% RSLogix 500 project traffic_light_rtc.RSS, saved by version 8.30.00.16 %
PROJECT "UNTITLED"    % processor: Bul.1763 MicroLogix 1100 Series A %

PROGRAM FILES
  LAD 2   7 rungs

DATA FILES
  O0 OUTPUT  4 elements
  I1 INPUT  6 elements
  S2 STATUS  66 elements
  B3 BINARY  2 elements
  T4 TIMER  4 elements
  C5 COUNTER  1 elements
  R6 CONTROL  1 elements
  N7 INTEGER  1 elements
  F8 FLOAT  1 elements
  B235   1 elements
  L244   4 elements
  L245   6 elements
  N254   1 elements
  N255   14 elements

LADDER 2
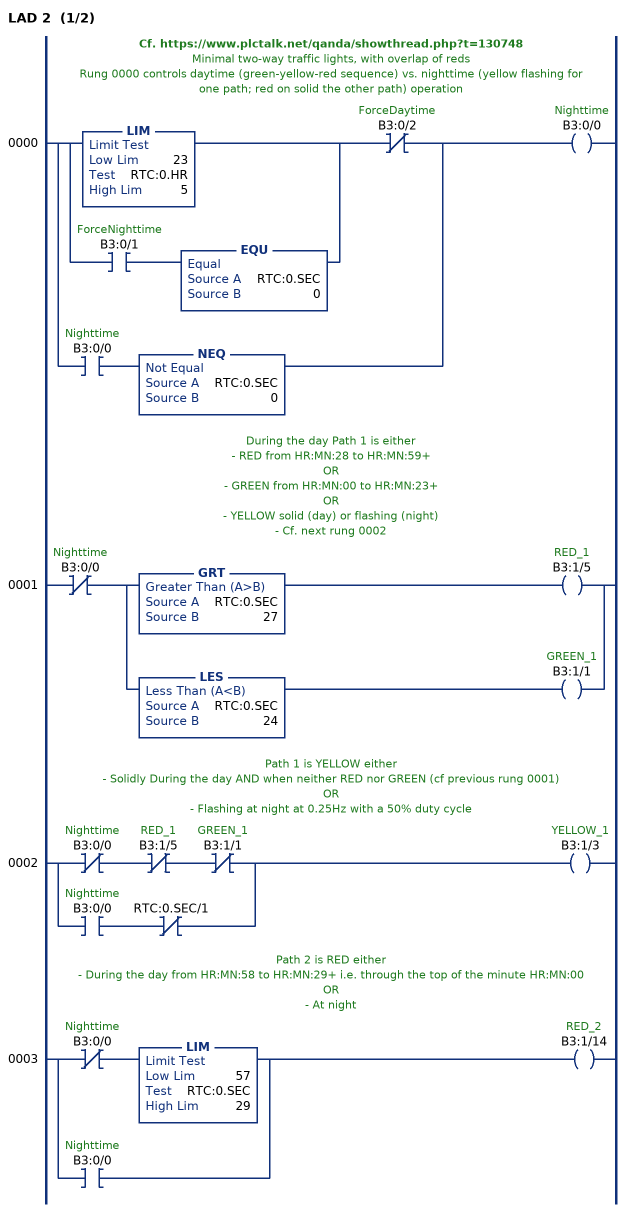
% Rung: 0 %
% TITLE: Cf. https://www.plctalk.net/qanda/showthread.php?t=130748 %
% Minimal two-way traffic lights, with overlap of reds
% Rung 0000 controls daytime (green-yellow-red sequence) vs. nighttime (yellow flashing for one path; red on solid the other path) operation %
SOR BST BST LIM 23 RTC:0.HR 5 NXB XIC B3:0/1 EQU RTC:0.SEC 0 BND XIO B3:0/2 NXB XIC B3:0/0 NEQ RTC:0.SEC 0 BND OTE B3:0/0 EOR
%   B3:0/1  "ForceNighttime" %
%   B3:0/2  "ForceDaytime" %
%   B3:0/0  "Nighttime" %
% Rung: 1 %
% During the day Path 1 is either
% - RED from HR:MN:28 to HR:MN:59+
% OR
% - GREEN from HR:MN:00 to HR:MN:23+
% OR
% - YELLOW solid (day) or flashing (night)
%   - Cf. next rung 0002 %
SOR XIO B3:0/0 BST GRT RTC:0.SEC 27 OTE B3:1/5 NXB LES RTC:0.SEC 24 OTE B3:1/1 BND EOR
%   B3:0/0  "Nighttime" %
%   B3:1/5  "RED_1" %
%   B3:1/1  "GREEN_1" %
% Rung: 2 %
% Path 1 is YELLOW either
% - Solidly During the day AND when neither RED nor GREEN (cf previous rung 0001)
% OR
% - Flashing at night at 0.25Hz with a 50% duty cycle %
SOR BST XIO B3:0/0 XIO B3:1/5 XIO B3:1/1 NXB XIC B3:0/0 XIO RTC:0.SEC/1 BND OTE B3:1/3 EOR
%   B3:0/0  "Nighttime" %
%   B3:1/5  "RED_1" %
%   B3:1/1  "GREEN_1" %
%   B3:1/3  "YELLOW_1" %
% Rung: 3 %
% Path 2 is RED either
% - During the day from HR:MN:58 to HR:MN:29+ i.e. through the top of the minute HR:MN:00
% OR
% - At night %
SOR BST XIO B3:0/0 LIM 57 RTC:0.SEC 29 NXB XIC B3:0/0 BND OTE B3:1/14 EOR
%   B3:0/0  "Nighttime" %
%   B3:1/14  "RED_2" %

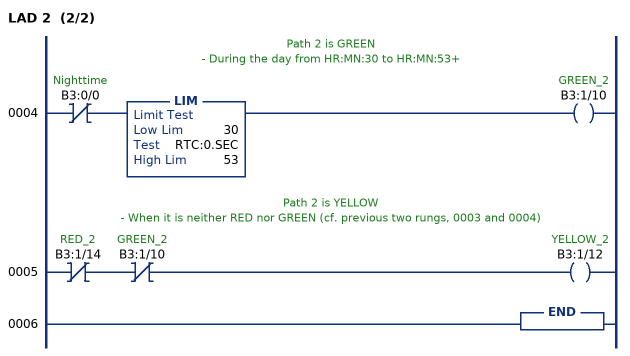
% Rung: 4 %
% Path 2 is GREEN
% - During the day from HR:MN:30 to HR:MN:53+ %
SOR XIO B3:0/0 LIM 30 RTC:0.SEC 53 OTE B3:1/10 EOR
%   B3:0/0  "Nighttime" %
%   B3:1/10  "GREEN_2" %
% Rung: 5 %
% Path 2 is YELLOW
% - When it is neither RED nor GREEN (cf. previous two rungs, 0003 and 0004) %
SOR XIO B3:1/14 XIO B3:1/10 OTE B3:1/12 EOR
%   B3:1/14  "RED_2" %
%   B3:1/10  "GREEN_2" %
%   B3:1/12  "YELLOW_2" %
% Rung: 6 %
SOR END EOR

DATA TABLE (non-zero values as saved)
DATA T4
% .PRE .ACC %
% T4:0 % 30 0
% T4:1 % 25 0
% T4:2 % 5 0
% T4:3 % 25 0
DATA R6
% .LEN .POS %
% R6:0 % 128 0
